{attribute 'GeneratedUsingTerminal: EK1100-0000-0018'}
{attribute addProperty BoxType "EK1100-0000-0018"}
{attribute addProperty Id "Beckhoff_EP4xxxEK1122Beckhoff_EP4xxxEK1122_F9FB0855336"}
{attribute addProperty CRC "1007397806"}
{attribute addProperty Size "336"}
TYPE Beckhoff_EP4xxx_3C0BABAE EXTENDS EK1100_AB5A9467 :
STRUCT
	{attribute addProperty Name "Beckhoff_EP4xxxEK1122"}
	{attribute addProperty PreviousPort "Beckhoff EP4xxx : B"}
	Beckhoff_EP4xxxEK1122 : Beckhoff_EP4xxxEK1122_F9FB0855;
END_STRUCT
END_TYPE

(* stored: Version 1.2.0.0, ProductVersion 3.1.4024.9
   DUT Beckhoff_EP4xxx_3C0BABAE: Id {dd2191b4-c6e3-4782-b133-f234a343fe5a} *)
